FUNCTION AnyToString : T_MaxString
VAR_INPUT
	a : ANY;
END_VAR

AnyToString := AnyTypeToString(a);

END_FUNCTION

(* stored: Version 1.1.0.1
   POU AnyToString: Id {1f0f5a07-7468-0acf-0462-c5684b77e674}, SpecialFunc None *)
